// TIA Portal V16 export
// export: Created 2025-12-18T09:29:18.5098521Z, ExportSetting WithDefaults, DisplayName Totally Integrated Automation Portal, DisplayVersion V16, DisplayName TIA Portal Version Control Interface, DisplayVersion V16, DisplayName TIA Portal Openness, DisplayVersion V16, DisplayName STEP 7 Professional, DisplayVersion V16, DisplayName STEP 7 Safety, DisplayVersion V16, DisplayName WinCC Advanced, DisplayVersion V16
VAR_GLOBAL   // PLC tag table "Inputs"
   iIO_xS1EntrySensor AT %I0.1 : Bool;
   iIO_xS1ExitSensor AT %I0.2 : Bool;
   iIO_xS1PositionerSensor AT %I0.3 : Bool;
   iIO_xS1ClampSensor AT %I0.4 : Bool;
   iIO_xS2EntrySensor AT %I0.5 : Bool;
   iIO_xS2ExitSensor AT %I0.6 : Bool;
   iIO_xS2PositionerSensor AT %I0.7 : Bool;
   iIO_xS2ClampSensor AT %I1.0 : Bool;
   iIO_xS3EntrySensor AT %I1.1 : Bool;
   iIO_xS3ExitSensor AT %I1.2 : Bool;
   iIO_xS3PositionerSensor AT %I1.3 : Bool;
   iIO_xS3ClampSensor AT %I1.4 : Bool;
   iIO_xS1ResetButton AT %I1.5 : Bool;
   iIO_xSupplyExitSensor AT %I0.0 : Bool;
   iIO_xS1EmergencyButton AT %I1.6 : Bool;
   iIO_xS2ResetButton AT %I2.0 : Bool;
   iIO_xS2EmergencyButton AT %I2.1 : Bool;
   iIO_xS3ResetButton AT %I2.2 : Bool;
   iIO_xS3EmergencyButton AT %I2.3 : Bool;
   iIO_xSupplyEntrySensor AT %I1.7 : Bool;
END_VAR
